// TIA Portal V16 export
// export: Created 2023-01-04T15:44:09.016548Z, ExportSetting WithDefaults, DisplayName Totally Integrated Automation Portal, DisplayVersion V16, DisplayName TIA Portal Version Control Interface, DisplayVersion V16, DisplayName TIA Portal Openness, DisplayVersion V16, DisplayName STEP 7 Professional, DisplayVersion V16, DisplayName STEP 7 Safety, DisplayVersion V16, DisplayName WinCC Advanced, DisplayVersion V16
FUNCTION_BLOCK "Operation_cycle"   // FB8, LAD
{ S7_Optimized_Access := 'TRUE' }
VERSION : 0.1
// stored: AutoNumber true, IsIECCheckEnabled false, IsRetainMemResEnabled false, MemoryReserve 100, SetENOAutomatically false, UDAEnableTagReadback false
   VAR
      begun : Bool;
   END_VAR
   VAR_TEMP   // added for the SCL form of the ladder/FBD networks
      _w1 : Bool;
      _w2 : Bool;
      _w3 : Bool;
   END_VAR
BEGIN

REGION Network 1
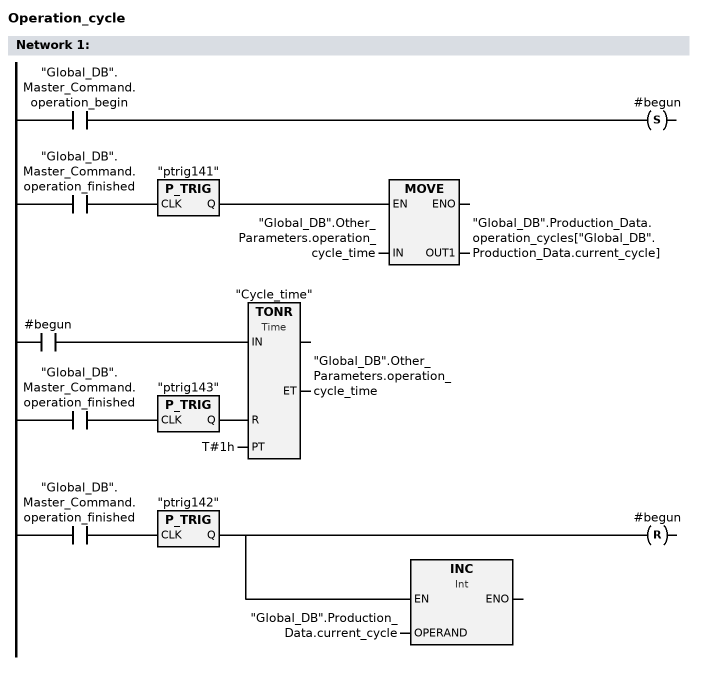
   RUNG wire#powerrail
      Contact( "Global_DB".Master_Command.operation_begin )
      S_Coil( #begun )
   END_RUNG
   RUNG wire#powerrail
      Contact( "Global_DB".Master_Command.operation_finished )
      P_Trig( "ptrig141" )
      Move(in := "Global_DB".Other_Parameters.operation_cycle_time, out1 => "Global_DB".Production_Data.operation_cycles["Global_DB".Production_Data.current_cycle])
   END_RUNG
   RUNG wire#powerrail
      Contact( #begun )
      { S7_Templates := "time_type := Time" } "Cycle_time".TONR(r := wire#w1, pt := T#1h, et => "Global_DB".Other_Parameters.operation_cycle_time)
   END_RUNG
   RUNG wire#powerrail
      Contact( "Global_DB".Master_Command.operation_finished )
      P_Trig( "ptrig143" )
   END_RUNG wire#w1
   RUNG wire#powerrail
      Contact( "Global_DB".Master_Command.operation_finished )
      P_Trig( "ptrig142" )
      wire#w2
      R_Coil( #begun )
   END_RUNG
   RUNG wire#w2
      { S7_Templates := "DestType := Int" } Inc( "Global_DB".Production_Data.current_cycle )
   END_RUNG
   // the same network as SCL:
   IF "Global_DB".Master_Command.operation_begin THEN #begun := TRUE; END_IF;
   #_w1 := "Global_DB".Master_Command.operation_finished AND NOT "ptrig141";   // rising edge
   "ptrig141" := "Global_DB".Master_Command.operation_finished;
   IF #_w1 THEN
       "Global_DB".Production_Data.operation_cycles["Global_DB".Production_Data.current_cycle] := "Global_DB".Other_Parameters.operation_cycle_time;
   END_IF;
   #_w2 := "Global_DB".Master_Command.operation_finished AND NOT "ptrig143";   // rising edge
   "ptrig143" := "Global_DB".Master_Command.operation_finished;
   "Cycle_time".TONR(IN := #begun,
                     R := #_w2,
                     PT := T#1h,
                     ET => "Global_DB".Other_Parameters.operation_cycle_time);
   #_w3 := "Global_DB".Master_Command.operation_finished AND NOT "ptrig142";   // rising edge
   "ptrig142" := "Global_DB".Master_Command.operation_finished;
   IF #_w3 THEN
       #begun := FALSE;
       "Global_DB".Production_Data.current_cycle := "Global_DB".Production_Data.current_cycle + 1;
   END_IF;
END_REGION
END_FUNCTION_BLOCK
